// TIA Portal V20 export
// export: Created 2025-12-01T14:57:17.2763778Z, ExportSetting None, DisplayName Totally Integrated Automation Portal, DisplayVersion V20 Update 3, DisplayName TIA Portal Openness, DisplayVersion V20 Update 3, DisplayName TIA Portal Version Control Interface, DisplayVersion V20 Update 3, DisplayName STEP 7 Professional, DisplayVersion V20 Update 3, DisplayName STEP 7 Safety, DisplayVersion V20 Update 2, DisplayName WinCC Basic/Comfort/Advanced, DisplayVersion V20 Update 3, DisplayName WinCC Professional, DisplayVersion V20 Update 3, DisplayName WinCC Unified, DisplayVersion V20 Update 3
DATA_BLOCK "DB934_Datos_VarOmronMX2_V2"   // DB934
{ S7_Optimized_Access := 'FALSE' }
AUTHOR : OMRON
NAME : 20130412
VERSION : 3.0
// stored: AutoNumber false
   VAR
      Red_01 { S7_SetPoint := 'True'} : Array[1..126] of "UDT_VarOmronMX2_V2";   // Red 01 de Variadores Omron MX2
      Red_02 { S7_SetPoint := 'True'} : Array[1..126] of "UDT_VarOmronMX2_V2";   // Red 02 de Variadores Omron MX2
   END_VAR
BEGIN
END_DATA_BLOCK
